FUNCTION F_SaveExceptionCode
VAR_INPUT
	excInput : __SYSTEM.ExceptionCode;
END_VAR

IF GVL_Exceptions.nExcIndex <= GVL_Exceptions.cMaxExc THEN
    GVL_Exceptions.aExceptionHistory[GVL_Exceptions.nExcIndex] := excInput;
    GVL_Exceptions.nExcIndex := GVL_Exceptions.nExcIndex + 1;
END_IF

END_FUNCTION

(* stored: Version 1.1.0.1, ProductVersion 3.1.4024.12
   POU F_SaveExceptionCode: Id {8ffa827d-75e0-4a59-a2d0-1004c18d2202}, SpecialFunc None *)
